FUNCTION_BLOCK TmsEmbarkStation IMPLEMENTS I_Station, I_Cyclic, I_Resettable, I_Object
VAR
	_IsClear : BOOL := TRUE;
	_Complete : BOOL;
	_Operating : BOOL;
	_Ready : BOOL := TRUE;
	_Position : LREAL := 0.0;
	_HasMover : BOOL;
	MoverArrive : R_TRIG;
	_MyMover : I_XtsMover;
	SwitchAxisPosCtrl : I_Lift;
	_Track1SwitchPosition : MC_LREAL;
	_Track2SwitchPosition : MC_LREAL;
	ExecuteSequence : BOOL;
	_MyTrackNumber : INT := 1;
	_State : EmbarkStationStates;
	_MoverTravelPosition : MC_LREAL;
	_BoardVelocity : MC_LREAL := 100.0;
	_SwitchVelocity : MC_LREAL := 200.0;
	_MoverLeavePosition : LREAL;
	Called : BOOL;
END_VAR

{analysis -2}

PROPERTY BoardVelocity : MC_LREAL
GET
BoardVelocity := _BoardVelocity;
END_GET
SET
_BoardVelocity := BoardVelocity;
END_SET
END_PROPERTY

METHOD Cycle : HRESULT
MoverArrive(CLK := _HasMover);
IF MoverArrive.Q THEN
	_IsClear := FALSE;
	_Ready := FALSE;
	_Operating := TRUE;
	_Complete := FALSE;
END_IF
Operation();
END_METHOD

(*FB_Init is always available implicitly and it is used primarily for initialization.
The return value is not evaluated. For a specific influence, you can also declare the
methods explicitly and provide additional code there with the standard initialization
code. You can evaluate the return value.*)
METHOD FB_Init : BOOL
VAR_INPUT
	(* TRUE: the retain variables are initialized (reset warm / reset cold)*)
	bInitRetains	: BOOL;
	(* TRUE: the instance will be copied to the copy code afterward (online change)   *)
	bInCopyCode	: BOOL;
	Position	: LREAL;
	SwitchAxis : I_Lift;
	MyTrackNumber : INT;
	Track1SwitchPosition : LREAL;
	Track2SwitchPsoition : LREAL;
	MoverOnSwitchPosition : LREAL;
END_VAR
_Position := Position;
SwitchAxisPosCtrl := SwitchAxis;
_MyTrackNumber := MyTrackNumber;
_Track1SwitchPosition := Track1SwitchPosition;
_Track2SwitchPosition := Track2SwitchPsoition;
_MoverTravelPosition := moverOnSwitchPosition;
END_METHOD

METHOD HasMover : BOOL
HasMover := _HasMover;
END_METHOD

METHOD IsClear : BOOL
IsClear := _IsClear;
END_METHOD

METHOD isComplete : BOOL
isComplete := _Complete;
END_METHOD

METHOD IsOperating : BOOL
IsOperating := _Operating;
END_METHOD

METHOD IsReady : BOOL
IsReady := _Ready;
END_METHOD

METHOD MyMover : HRESULT
VAR_INPUT
	mover	: I_XtsMover;
END_VAR
IF mover = 0 THEN
	MyMover := -1;
	RETURN;
END_IF
IF _HasMover THEN
	MyMover := -2;
	RETURN;
END_IF
_HasMover := TRUE;
_MyMover := mover;
END_METHOD

METHOD Operation : BOOL
VAR_INPUT
END_VAR
CASE _State OF
	EmbarkStationStates.Init:
		_Operating := _IsClear := _Complete := _Ready := _HasMover := FALSE;
		_State := EmbarkStationStates.Ready;
	
	EmbarkStationStates.Ready:	
		IF ExecuteSequence THEN
			_Operating := _Complete := _HasMover := FALSE;
			_IsClear := _Ready := TRUE;
			_State := EmbarkStationStates.Waiting;
		END_IF
	
	EmbarkStationStates.Waiting:
		IF _HasMover THEN
			_State := EmbarkStationStates.HasSwitch;
			_Operating := TRUE;
			_IsClear := FALSE;
			_Ready := FALSE;
			_Complete := FALSE;
		END_IF
	
	EmbarkStationStates.HasSwitch:
		IF ((_MyTrackNumber = 1 AND SwitchAxisPosCtrl.isAtPosition(_Track1SwitchPosition))
			OR (_MyTrackNumber = 2 AND SwitchAxisPosCtrl.isAtPosition(_Track2SwitchPosition))) AND NOT SwitchAxisPosCtrl.Assigned THEN
				SwitchAxisPosCtrl.Assigned := TRUE;
				_State := EmbarkStationStates.Boarding;
		ELSIF NOT Called THEN
			_State := EmbarkStationStates.Call;
		END_IF	
		
	EmbarkStationStates.Call:
		IF NOT SwitchAxisPosCtrl.Assigned AND_THEN SwitchAxisPosCtrl.IsStationary() THEN
			IF _MyTrackNumber = 1 THEN
				SwitchAxisPosCtrl.Call(Position := _Track1SwitchPosition, Velocity := _SwitchVelocity);
			ELSE
				SwitchAxisPosCtrl.Call(Position := _Track2SwitchPosition, Velocity := _SwitchVelocity);
			END_IF
			SwitchAxisPosCtrl.Assigned := TRUE;
			Called := TRUE;
			_State := EmbarkStationStates.test;
		END_IF
		
	EmbarkStationStates.test:
		IF (_MyTrackNumber = 1 AND SwitchAxisPosCtrl.isAtPosition(_Track1SwitchPosition))
			OR (_MyTrackNumber = 2 AND SwitchAxisPosCtrl.isAtPosition(_Track2SwitchPosition)) THEN
				_State := EmbarkStationStates.Boarding;
				Called := FALSE;
		END_IF	
		
	EmbarkStationStates.Boarding:
		_MyMover.MoveTo(RequiredPosition := _MoverTravelPosition, MoveVelocity := _BoardVelocity, NonModuloMove := FALSE);
		IF _MoverTravelPosition > _MyMover.GetActiveTrackLength() THEN
			IF (_MyMover.ActualTrackPosition > (_MoverTravelPosition - _MyMover.GetActiveTrackLength()) - 0.3 
				AND _MyMover.ActualTrackPosition < (_MoverTravelPosition - _MyMover.GetActiveTrackLength()) + 0.3) THEN
				_State := EmbarkStationStates.BoardingComplete;
			END_IF
		ELSE
			IF (_MyMover.ActualTrackPosition > _MoverTravelPosition - 0.3 AND _MyMover.ActualTrackPosition < _MoverTravelPosition + 0.3) THEN
				_State := EmbarkStationStates.BoardingComplete;
			END_IF
		END_IF
		
	EmbarkStationStates.BoardingComplete:
		IF _MyTrackNumber = 1 THEN
			SwitchAxisPosCtrl.MoveToPosition(Position := _Track2SwitchPosition, Velocity := _SwitchVelocity);
		ELSE
			SwitchAxisPosCtrl.MoveToPosition(Position := _Track1SwitchPosition, Velocity := _SwitchVelocity);
		END_IF
		_State := EmbarkStationStates.Moving;
		
	EmbarkStationStates.Moving:
		IF (_MyTrackNumber = 1 AND SwitchAxisPosCtrl.isAtPosition(position := _Track2SwitchPosition)) OR
			(_MyTrackNumber = 2 AND SwitchAxisPosCtrl.isAtPosition(position := _Track1SwitchPosition)) THEN
			_State := EmbarkStationStates.ActivateTrackForMover;
		END_IF
		
	EmbarkStationStates.ActivateTrackForMover:
		IF _MyTrackNumber = 1 THEN
			IF SUCCEEDED(_MyMover.ActivateTrack(Track := 2)) THEN
				_State := EmbarkStationStates.CheckActiveTrack;
			END_IF
		ELSE
			IF SUCCEEDED(_MyMover.ActivateTrack(Track := 1)) THEN
				_State := EmbarkStationStates.CheckActiveTrack;
			END_IF
		END_IF
		
	EmbarkStationStates.CheckActiveTrack:
		IF _MyTrackNumber = 1 AND_THEN _MyMover.MoversActiveTrack = 2 THEN
			_State := EmbarkStationStates.CheckMoverLeft;
			_MoverLeavePosition := _MyMover.AxisRef.NcToPlc.ActPos;
		ELSIF  _MyMover.MoversActiveTrack = 1 THEN
			_State := EmbarkStationStates.CheckMoverLeft;
			_MoverLeavePosition := _MyMover.AxisRef.NcToPlc.ActPos;
		END_IF
	
	EmbarkStationStates.CheckMoverLeft:
		_Complete := TRUE;
		IF _MyMover.AxisRef.NcToPlc.ActPos > _MoverLeavePosition + 100 THEN
			_State := EmbarkStationStates.Done;
			_HasMover := FALSE;
			SwitchAxisPosCtrl.Assigned := FALSE;
		END_IF
			
	EmbarkStationStates.Done:
		IF _Complete AND NOT _HasMover THEN
			_Operating := FALSE;
			_IsClear := TRUE;
			_Ready := TRUE;
			_State := EmbarkStationStates.Waiting;
		END_IF	
END_CASE
END_METHOD

PROPERTY Position : MC_LREAL
GET
Position := _Position;
END_GET
END_PROPERTY

METHOD RegisterWithParent
VAR_INPUT
	Parent	: Base_Library.I_HostObjects;
END_VAR
END_METHOD

METHOD Reset : HRESULT
_Complete := FALSE;
_IsClear := TRUE;
_Operating := FALSE;
_Ready := TRUE;
_HasMover := FALSE;
_State := EmbarkStationStates.Init;
SwitchAxisPosCtrl.Assigned := FALSE;
END_METHOD

METHOD StartSwitch : BOOL
VAR_INPUT
END_VAR
ExecuteSequence := TRUE;
END_METHOD

METHOD StopSwitch : BOOL
VAR_INPUT
END_VAR
ExecuteSequence := FALSE;
END_METHOD

PROPERTY SwitchVelocity : LREAL
GET
SwitchVelocity := _SwitchVelocity;
END_GET
SET
_SwitchVelocity := SwitchVelocity;
END_SET
END_PROPERTY

END_FUNCTION_BLOCK

(* stored: Version 1.1.0.1
   POU TmsEmbarkStation: Id {4d15a973-29cb-4ffe-934a-8f072d992ec0}, SpecialFunc None
   Folder Status: Id {fc30821c-889b-457b-acd5-7e0794e2da97}
   Property BoardVelocity: Id {af5577ef-90f6-4070-9e3d-dce62d068c94}
   Get Get: Id {442f20d9-4d5c-462e-ace0-37721614361e}
   Set Set: Id {4f476cb8-1c36-46ee-b33f-8098bec190be}
   Method Cycle: Id {3f7d84b9-4220-4895-8d1f-d1319db89048}
   Method FB_Init: Id {c56e5d7e-44de-4ea5-9429-5a143178668d}
   Method HasMover: Id {01ba8fbd-2454-4e68-9b4a-9db0f953212c}
   Method IsClear: Id {43301cfc-5dfe-497a-ba25-2baea0d242aa}
   Method isComplete: Id {44421f60-5729-4d12-9b71-06a85fd9d019}
   Method IsOperating: Id {df31fe6f-4d2e-47a8-9a3f-cb59b84fd3a0}
   Method IsReady: Id {ecaac7cf-e1f3-4b8e-82e7-477bdefe5978}
   Method MyMover: Id {53ce83f8-f376-4c29-a057-798a57ce6dc6}
   Method Operation: Id {79e49ccb-98b2-4f0a-86f7-22dcc9a5dd9a}
   Property Position: Id {57781d24-723f-4dbc-b59b-493697f347b8}
   Get Get: Id {846aa0af-3762-492c-8088-91ff454623be}
   Method RegisterWithParent: Id {ae1250b4-e8d3-4bd2-8110-48d016d30ba8}
   Method Reset: Id {95aecf88-84d1-40dd-83f3-696248ea5185}
   Method StartSwitch: Id {c29e9395-8979-4e9a-90a8-1d97909d0ac9}
   Method StopSwitch: Id {3cacf78b-01e4-4c36-b301-1826803c65db}
   Property SwitchVelocity: Id {2b2ab201-99a2-4b79-87da-05eb4b2bdaf0}
   Get Get: Id {cd238776-2665-438e-8843-6901647c425c}
   Set Set: Id {3a523177-e66f-47d0-8004-3fc4fbb2e246} *)
